TYPE ASCII :
STRUCT	
	AscByte			:ARRAY[1..5] OF BYTE;
END_STRUCT
END_TYPE

(* stored: Version 1.1.0.1, ProductVersion 3.1.4024.2
   DUT ASCII: Id {76ed04be-f1c7-461e-bf80-0a90c901315e} *)
